// TIA Portal V15 export
// export: Created 2018-05-29T12:25:38.1552518Z, ExportSetting WithDefaults, DisplayName Totally Integrated Automation Portal, DisplayVersion V15, DisplayName STEP 7 Professional, DisplayVersion V15, DisplayName WinCC Professional, DisplayVersion V15, DisplayName TIA Portal Openness, DisplayVersion V15
FUNCTION "EM_Instance_4_fc" : Void   // FC1, STL
TITLE = _fc
{ S7_Optimized_Access := 'TRUE' }
VERSION : 0.1
// test
// stored: AutoNumber true, UDAEnableTagReadback false
BEGIN

NETWORK
TITLE = Main
// comment:


// Call the EM FB with the corresponding DB instance
      CALL  "EM_I_OUT", "EM_Instance_4"
      ( sampletime       := ,
        em_id            := #"29",
        Request          := ,
        Command          := ,
        Pressure_SP      := ,
        Pump_RUN         := #"M103.QNOFF2",
        Pump_QERR        := #"M103.QERR",
        Pump_EERR        := #"M103.QERR_EXT",
        FS01_PV          := #"LS002.QON",
        PIC01_PV         := #"LIC004.PV",
        PIC01_ERR        := #"LIC004.QERR",
        LT01_PV          := #"LT004.QfVal",
        LT01_AHH         := #"LT004.LIM_Qb01",
        LT01_AH          := #"LT004.LIM_Qb02",
        LT01_AL          := #"LT004.LIM_Qb03",
        LT01_ALL         := #"LT004.LIM_Qb04",
        LT01_ERR         := #"LT004.QERR",
        XV_Bottom_OPN    := ,
        XV_Bottom_CLS    := ,
        XV_Bottom_MERR   := ,
        BV_Bottom_OPN    := #"MV004.QOPEN",
        BV_Bottom_CLS    := #"MV004.QCLOSE",
        BV_Bottom_MERR   := #"MV004.QMON_ERR",
        BV_Tran_M04_OPN  := #"MV003.QOPEN",
        BV_Tran_M04_CLS  := #"MV003.QCLOSE",
        BV_Tran_M04_MERR := #"MV003.QMON_ERR",
        steptime_s       := ,
        steptime_m       := ,
        steptime_h       := ,
        first_scan       := ,
        last_scan        := ,
        error_index_db   := ,
        Owner            := ,
        Status           := ,
        CM_error         := ,
        CM_error_no      := ,
        q_bACTVIE        := ,
        Level            := ,
        Pressure         := ,
        Pump_ON          := #"M103.L_ON",
        Pump_AUT         := #"M103.L_AUT",
        PIC01_EXT        := #"LIC004.L_REMOTE",
        PIC01_SP         := #"LIC004.HMI_SP_INT",
        PIC01_AUT        := #"LIC004.L_AUT",
        PIC01_VAL_OUT    := #"LIC004.HMI_MAN",
        PIC01_SET_SP     := #"LIC004.Set_SP",
        PIC01_SET_OUT    := #"LIC004.Set_Output",
        XV_Bottom_CMD    := ,
        BV_Bottom_CMD    := #"MV004.AUT_OP",
        BV_Tran_M04_CMD  := #"MV003.AUT_OP"
      );
END_FUNCTION
